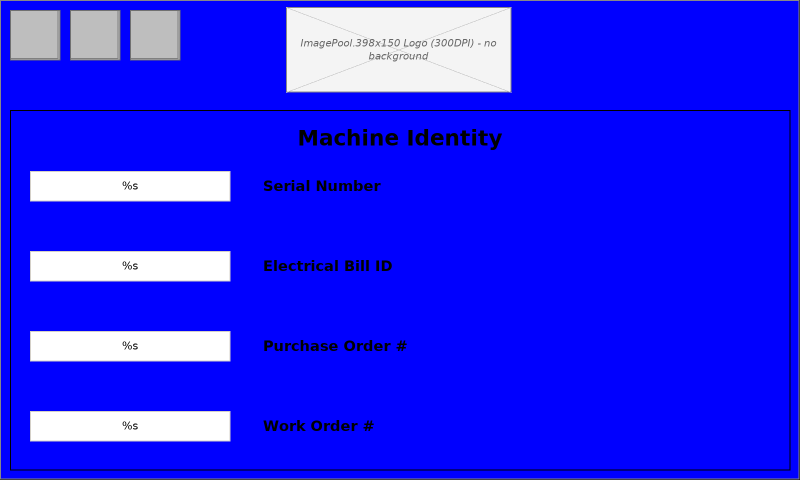
VISUALIZATION Machine_ID_Settings  // 800x480
    Rectangle (0,0 800x480)
    Rectangle (10,110 780x360)
    Textfield (30,171 200x30), "%s", text variable: GVL.Machine_Serial_Number
        OnMouseClick: write the text variable via VisuDialogs.Keypad
    Textfield (30,251 200x30), "%s", text variable: GVL.Electrical_Bill_ID
        OnMouseClick: write the text variable via VisuDialogs.Keypad
    Textfield (30,331 200x30), "%s", text variable: GVL.Purchase_Order_Number
        OnMouseClick: write the text variable via VisuDialogs.Keypad
    Image (286,7 225x85), image: ImagePool.398x150 Logo (300DPI) - no background
        OnMouseClick: change screen: Home
    Button (70,10 50x50), image: VisuSymbols.Symbols.Home
        OnMouseClick: change screen: Home
    Label (0,120 800x36), "Machine Identity"
    Button (10,10 50x50), image: VisuSymbols.Symbols.TriangleLeft
        OnMouseClick: change screen: Previous Home
    Textfield (30,411 200x30), "%s", text variable: GVL.Work_Order_Number
        OnMouseClick: write the text variable via VisuDialogs.Keypad
    Label (260,171 225x30), "Serial Number"
    Label (260,251 225x30), "Electrical Bill ID"
    Label (260,331 225x30), "Purchase Order #"
    Label (260,411 225x30), "Work Order #"
    Label (550,331 225x30)
    Button (130,10 50x50), image: VisuSymbols.Symbols.TwoWheels
        OnMouseClick: change screen: Settings_Menu
END_VISUALIZATION

(* stored: Version 1.1.0.1, ProductVersion 3.1.4024.12
   Visu Machine_ID_Settings: Id {0b78f58f-99fe-4ba3-90de-779aec4eb209} *)
